{attribute 'qualified_only'}
{attribute 'strict'}
TYPE E_Light :
(
	Green,
	Red
);
END_TYPE

(* stored: Version 1.1.0.1, ProductVersion 3.1.4024.12
   DUT E_Light: Id {1de47428-7906-4d90-9b1f-2cf4422e48c4} *)
